FUNCTION_BLOCK FB_VectorCrossProduct_Test EXTENDS FB_TestSuite
VAR_INPUT
END_VAR
VAR_OUTPUT
END_VAR
VAR
END_VAR

WhenWrongSizeExpectError();
WhenMatchingSizeExpectResult();
WhenBackwardsExpectOppositeResult();

METHOD PRIVATE WhenBackwardsExpectOppositeResult
VAR_INPUT
END_VAR
VAR
	MV : DynamicMatrix;
	V1 : DynamicMatrix;
	V2 : DynamicMatrix;
	V3 : DynamicMatrix;
	Vs : ARRAY[0..1] OF POINTER TO MAtrix;
	M1 : DynamicMatrix;
	Result : BOOL;
END_VAR
TEST('WhenBackwardsExpectOppositeResult');

// @TEST-RUN
Vs[1] := ADR(V1);
Vs[0] := ADR(V2);

MV.InitIdentity(3);
V1.AsColVector(MV,0);
V2.AsColVector(MV,1);
V3.AsColVector(MV,2);
V3.Scale(-1);

Result := M1.AsVectorCrossProduct(Vs);

// @TEST-ASSERT
AssertTrue(Result,'Main function call was not successful');
AssertTrue(M1.IsEqual(V3),'Result is the correct vector');

TEST_FINISHED();
END_METHOD

METHOD PRIVATE WhenMatchingSizeExpectResult
VAR_INPUT
END_VAR
VAR
	MV : DynamicMatrix;
	V1 : DynamicMatrix;
	V2 : DynamicMatrix;
	V3 : DynamicMatrix;
	Vs : ARRAY[0..1] OF POINTER TO MAtrix;
	M1 : DynamicMatrix;
	Result : BOOL;
END_VAR
TEST('WhenMatchingSizeExpectResult');

// @TEST-RUN
Vs[0] := ADR(V1);
Vs[1] := ADR(V2);

MV.InitIdentity(3);
V1.AsColVector(MV,0);
V2.AsColVector(MV,1);
V3.AsColVector(MV,2);

Result := M1.AsVectorCrossProduct(Vs);

// @TEST-ASSERT
AssertTrue(Result,'Main function call was not successful');
AssertTrue(M1.IsEqual(V3),'Result is not the correct vector');

TEST_FINISHED();
END_METHOD

METHOD PRIVATE WhenWrongSizeExpectError
VAR_INPUT
END_VAR
VAR
	V1 : DynamicMatrix;
	V2 : DynamicMatrix;
	Vs : ARRAY [0..1] OF POINTER TO Matrix;
	M1 : DynamicMatrix;
	Result : BOOL;
END_VAR
TEST('WhenWrongSizeExpectError');

// @TEST-RUN
Vs[0] := ADR(V1);
Vs[1] := ADR(V2);

V1.InitVector(3,1,1);
V2.InitVector(4,1,1);

Result := Vector_CrossProduct(M1,Vs);

// @TEST-ASSERT
AssertFalse(Result,'Main function call was unexpectedly successful');

TEST_FINISHED();
END_METHOD

END_FUNCTION_BLOCK

(* stored: Version 1.1.0.1, ProductVersion 3.1.4024.9
   POU FB_VectorCrossProduct_Test: Id {27cbb6d0-ee82-05a0-0885-25c9ace8e002}, SpecialFunc None
   Method WhenBackwardsExpectOppositeResult: Id {c4adfab1-3c64-086f-0455-f78b963aca2f}
   Method WhenMatchingSizeExpectResult: Id {210123e9-79aa-07ab-204d-1d5b02cf36e9}
   Method WhenWrongSizeExpectError: Id {94f8a6a5-daf1-0562-3890-919c18f161b5} *)
